PROGRAM MAIN
VAR
	
	
	stAxis				: ARRAY[1..2] OF AXIS_REF;
	fbMcPower			: ARRAY[1..2] OF MC_Power;
	fbMcReset			: ARRAY[1..2] OF MC_Reset;
	fbMcMoveVelocity	: ARRAY[1..2] OF MC_MoveVelocity;
	fbMcHalt			: ARRAY[1..2] OF MC_Halt;
	
	bPower		: BOOL;
	bRun		: BOOL;
	bStop		: BOOL;
	bMcReset		AT%I*	: BOOL;
	bSafetyReset	AT%Q*	: BOOL;
	bSafetyRun		AT%Q*	: BOOL := TRUE;
	bSafetyErrAck	AT%Q*	: BOOL;
	diSpeedAct		AT%Q*	: DINT;
	diSpeedCmd		AT%Q*	: DINT; 
	
	bWarningSigna0l		AT%I*	: BOOL;
	bWarningSigna02		AT%I*	: BOOL;
	Enc2ActError		AT%I*	: BOOL;
	Enc2CmdError		AT%I*	: BOOL;
	
	lrOverride		: LREAL := 50;
	_override		: LREAL;
	lrVelocity		: LREAL := 360;
	lrGearRate		: LREAL := 10;
	lrIncrement		: LREAL := 1048576;
	lrWheelIncrement	:LREAL;
	lrExtEncoderIncrement		: LREAL := 1000;
	
	diTaskIdx			: DINT;
	udiCycletime		: UDINT;
	udiTimeIntervel		: UDINT;
	udiCycleCount		: UDINT;
	fbDelaySampling		: FB_DelaySampling;
	fbDelaySamplingSet	: FB_DelaySampling;
	
	diPositionAct			: DINT;
	diPositionBufferAct		: DINT;
	diPositionCmd			: DINT;
	diPositionBufferCmd		: DINT;
	
	Mode	: INT;
	i		: UINT;
	//_Mode	: INT;
	//mode_change_delay_timer	: TON := (PT := T#1S);
	
	safety_input_collision_sensor AT%I* : BOOL;
	safety_master_station_emo AT%I* : BOOL;
	safety_emo AT%I* : ARRAY [1..2] OF BOOL;
	
	running_startup_delapy : TON := (PT := T#1S);
	
	eap_export_information	AT%Q* : ARRAY [0..7] OF BOOL;
	
	monitor_speed_average : FB_MovingAverage;
	monitor_refspeed_average : FB_MovingAverage;
	monitor_setspeed_average : FB_MovingAverage;

	SafetyMonitorSpeed AT%I* : DINT;
	SafetyRefMonitorSpeed AT%I* : DINT;
	SafetyMonitorSetSpeed AT%I* : DINT;
	
END_VAR


// Set override speed to 25 while 1sec after motor starting up. Otherwise safety error would occured by speed differential watching.
running_startup_delapy(IN := stAxis[1].Status.Moving);
IF running_startup_delapy.Q THEN
	_override := lrOverride;
ELSE
	_override := 30.0;
END_IF

FOR i:=1 TO 2 DO
	stAxis[i].ReadStatus();
	fbMcPower[i](
	Axis:= stAxis[i], 
	Enable:= bPower, 
	Enable_Positive:= bPower, 
	Enable_Negative:= bPower,
	Override := _override);

	fbMcHalt[i](
		Axis:= stAxis[i], 
		Execute:= bStop, 
		Deceleration:= 3600);
	
	fbMcReset[i](
		Axis:= stAxis[i], 
		Execute:= bMcReset);
	
	fbMcMoveVelocity[i](
		Axis:= stAxis[i],
		Execute:= bRun,
		Velocity:= lrVelocity, 
		//Direction:= MC_Direction.MC_Negative_Direction, 
		BufferMode:= MC_BufferMode.MC_Aborting);	
END_FOR
fbMcMoveVelocity[1].Direction := MC_Direction.MC_Negative_Direction;
fbMcMoveVelocity[2].Direction := MC_Direction.MC_Positive_Direction;

bSafetyReset := bMcReset;
bSafetyErrAck := bMcReset;
IF bMcReset THEN
	Mode := AreaStatus.Safe;
END_IF

IF NOT bWarningSigna0l THEN
	Mode := AreaStatus.Warning_Level1;
	IF NOT bWarningSigna02 THEN
		Mode := AreaStatus.Warning_Level2;
	END_IF
ELSIF (stAxis[1].NcToPlc.ErrorCode <> 0) OR (stAxis[2].NcToPlc.ErrorCode <> 0) THEN
	Mode := AreaStatus.Hazard;
ELSE
	Mode := AreaStatus.Safe;
END_IF

CASE Mode OF

	AreaStatus.Safe:
						lrOverride := 50;	
						
	AreaStatus.Warning_Level1:
						lrOverride := 25;
						
	AreaStatus.Warning_Level2:
						lrOverride := 10;
						
	AreaStatus.Hazard:
						lrOverride := 0;
	
END_CASE


lrWheelIncrement := lrIncrement * lrGearRate / 360;
diPositionAct := LREAL_TO_DINT(-1 * stAxis[1].NcToPlc.ActPos * lrWheelIncrement / lrExtEncoderIncrement);
diSpeedAct := diPositionAct - diPositionBufferAct; 
diPositionCmd := LREAL_TO_DINT(-1 * stAxis[1].NcToPlc.SetPos * lrWheelIncrement / lrExtEncoderIncrement);
diSpeedCmd := diPositionCmd - diPositionBufferCmd; 

diTaskIdx := GETCURTASKINDEXEX();
IF diTaskIdx > 0 THEN
    udiCycleTime := _TaskInfo[diTaskIdx].CycleTime;
	udiCycleCount := (udiTimeIntervel*10000) / udiCycleTime;
END_IF
fbDelaySampling(udiDelaySampling:= udiCycleCount, diData:= diPositionAct, diOutData=> diPositionBufferAct);
fbDelaySamplingSet(udiDelaySampling:= udiCycleCount, diData:= diPositionCmd, diOutData=> diPositionBufferCmd);

// Alarm signal

IF AlarmManager.init THEN
	GVL.fb_alarm[AlarmList.emergency_stop]^.set_activate := NOT safety_master_station_emo OR NOT safety_emo[1] OR NOT safety_emo[2];
	GVL.fb_alarm[AlarmList.approach]^.set_activate := Mode = AreaStatus.Warning_Level1;
	GVL.fb_alarm[AlarmList.proximity]^.set_activate := Mode = AreaStatus.Warning_Level2;
	GVL.fb_alarm[AlarmList.collision]^.set_activate :=  stAxis[1].Status.Moving AND NOT safety_input_collision_sensor;
	GVL.fb_alarm[AlarmList.encoder_error]^.set_activate :=  bPower AND ( NOT Enc2ActError OR NOT Enc2CmdError );

	// Send state to CP6606 controller station
	FOR i := 0 TO 7 DO
		IF i < AlarmEventParam.ALARM_MAX_COUNT THEN
			eap_export_information[i] := GVL.fb_alarm[i + 1]^.bActive;
		END_IF
	END_FOR
	eap_export_information[5] := NOT stAxis[1].Status.Disabled;
	eap_export_information[6] := stAxis[1].Status.Moving;	
END_IF

monitor_speed_average(put := SafetyMonitorSpeed);
monitor_refspeed_average(put := SafetyRefMonitorSpeed);
monitor_setspeed_average(put := SafetyMonitorSetSpeed);

AlarmManager.reset_button_input := bMcReset;
AlarmManager();

END_PROGRAM

(* stored: Version 1.1.0.1
   POU MAIN: Id {51fb128e-0b29-449f-81b5-c1bdf5c46aab}, SpecialFunc None *)
